(* PLC project LMM.project, Inovance company InoProShop(V1.9.1.6) InoProShop(V1.9.1.6) *)
(* stored: creationDateTime 2026-07-22T21:08:52.4325602, modificationDateTime 2026-07-22T21:08:38.7942337 *)

VAR_GLOBAL  (* GVL *)
  StartBtn AT %IX1.6 : BOOL;  (* 【面板启动】AT %IX1.6 → HMI_xStart/HMI_xEnable（上升沿 STOP→RUN） *)
  StopBtn AT %IX1.4 : BOOL;  (* 【面板停止】AT %IX1.4 → HMI_xStop *)
  ResetBtn : BOOL;  (* 【面板复位】→ HMI_xStopHold3s（错误复位脉冲）；地址现场可另绑 *)
  EStop AT %IX0.4 : BOOL;  (* 【面板急停】AT %IX0.4 正常=TRUE 按下=FALSE → 直通 HMI_xEStop *)
  StopLamp AT %QX0.6 : BOOL;  (* 【停止指示灯】AT %QX0.6 ← Dev_xStop（停止/待机） *)
  StartLamp AT %QX0.7 : BOOL;  (* 【启动/运行指示灯】AT %QX0.7 ← Dev_xRun（正在运行） *)
  JogVel : REAL;  (* 面板点动速度 → 桥接到 HMI_rJogVel* *)
  JogFwd : BOOL;  (* 面板前进 → 按 X 模式映射到 Sync/Diff/独立点动+ *)
  JogBwd : BOOL;  (* 面板后退 → 按 X 模式映射到 Sync/Diff/独立点动- *)
  JogUp : BOOL;  (* 面板上 → HMI_xJogZPos *)
  JogDown : BOOL;  (* 面板下 → HMI_xJogZNeg *)
  JogRight : BOOL;  (* 面板右 → HMI_xJogYPos *)
  JogLeft : BOOL;  (* 面板左 → HMI_xJogYNeg *)
  JogClockAdd : BOOL;  (* 顺时针 *)
  JogClockMis : BOOL;  (* 逆时针 *)
  JogACC : REAL;  (* 点动加速度 → AxisCmd_rAcc *)
  JogDEC : REAL;  (* 点动减速度 → AxisCmd_rDec *)
  HomeReq : BOOL;  (* 面板回零 → HMI_xHomeReqY/Z *)
  CaliForReq : BOOL;  (* 重力标定 *)
  ClearBruch : BOOL;  (* 毛刷清洗 *)
  yLength : REAL;  (* 龙门跨距/Y长度设定 4..6m → HMI_rWheelBase *)
  HMI_xEStop : BOOL;  (* 【急停】TRUE=未按下(正常)；FALSE=急停按下。可按可松，锁存由Logic保持 *)
  HMI_xStop : BOOL;  (* 【设备停止】短按RUN→STOP；长按3s故障复位 *)
  HMI_xStopHold3s : BOOL;  (* 【停止长按满3s脉冲】清急停锁存+轴错误复位+下使能 *)
  HMI_xEnable : BOOL;  (* 【使能/启动别名】与HMI_xStart等效；上升沿STOP→RUN *)
  Dev_xError : BOOL;  (* 【内部故障态】 *)
  Dev_xRun : BOOL;  (* 【内部运行态】 *)
  Dev_xStop : BOOL;  (* 【内部停机态】 *)
  eDevState : INT;  (* 【废弃】不做控制；显示请用 HMI_eDevState 派生 *)
  HMI_xDevError : BOOL;  (* 【故障灯设备级】 *)
  HMI_xDevRun : BOOL;  (* 【运行灯】 *)
  HMI_xDevStop : BOOL;  (* 【停机灯】 *)
  HMI_eOpMode : INT;  (* 【运行方式】0手动 1自动；配合Run灯 *)
  HMI_eDevState : INT;  (* 【设备状态码】0=STOP 1=RUN 2=ERROR *)
  HMI_xStart : BOOL;  (* 【设备启动】瞬时；上升沿STOP→RUN *)
  HMI_xJogYPos : BOOL;  (* 【Y点动+】TRUE移动 FALSE暂停；受限位/Z忙 *)
  HMI_xJogYNeg : BOOL;  (* 【Y点动-】TRUE移动 FALSE暂停 *)
  HMI_xJogZPos : BOOL;  (* 【Z点动+】TRUE移动 FALSE暂停 *)
  HMI_xJogZNeg : BOOL;  (* 【Z点动-】TRUE移动 FALSE暂停 *)
  HMI_xJogRPos : BOOL;  (* 【R点动+】预留；M5未就绪无效 *)
  HMI_xJogRNeg : BOOL;  (* 【R点动-】预留 *)
  HMI_xHomeY : BOOL;  (* 【Y回零】电平/上升沿触发；或配合轴选择\r\n *)
  HMI_xHomeZ : BOOL;  (* 【Z回零】电平/上升沿触发；或配合轴选择\r\n *)
  HMI_xHomeR : BOOL;  (* 【R回零】电平/上升沿触发；或配合轴选择\r\n *)
  HMI_iHomeAxis : INT := 0;  (* 【回零轴选择】0无 1=Y 2=Z 3=R\r\n *)
  HMI_xHomeExec : BOOL;  (* 【回零执行】上升沿：对 HMI_iHomeAxis 选定轴启动回零\r\n *)
  HMI_rJogVelX : REAL := 0.4;  (* 【X点动速度】龙门X基速设定 *)
  AxisCmd_rSpinVel : REAL := 0.0;
  HMI_rJogVelR : REAL := 0.2;  (* 【R轴手动速度】 *)
  HMI_rSpinVel : REAL := 0.3;  (* 【X轴旋转速度】 *)
  HMI_rJogVelY : REAL := 0.4;  (* 【Y点动速度】 *)
  HMI_rJogVelZ : REAL := 0.4;  (* 【Z点动速度】 *)
  HMI_rWheelBase : REAL := 5.0;  (* 【龙门跨距=Y行程】单位m，合法范围4..6；自动Y走距用此值 *)
  xEStopLatched : BOOL;  (* 【急停锁存】按下急停置位；仅长按停止复位可清 *)
  xEnablePermit : BOOL;  (* 【废弃】已删除设备态许可互锁 *)
  xFaultAggregate : BOOL;  (* 【故障汇总】任轴Fault *)
  xIlk_BlockYPlus : BOOL;  (* 【联锁禁Y+】由Y+限位派生 *)
  xIlk_BlockYNeg : BOOL;  (* 【联锁禁Y-】由Y-限位派生 *)
  xIlk_BlockZPlus : BOOL;  (* 【联锁禁Z+】由Z+限位派生 *)
  xIlk_BlockZNeg : BOOL;  (* 【联锁禁Z-】由Z-限位派生 *)
  xIlk_BlockYWhenZ : BOOL;  (* 【Z动禁Y】Z运动中禁止Y点动 *)
  xM5Ready : BOOL := TRUE;  (* 【第5轴就绪】TRUE=启用 R(Axis_4)；FALSE=忽略R\r\n *)
  HMI_xLampEStop : BOOL;  (* 【急停灯】HMI读；锁存或按钮仍按下 *)
  HMI_xLampEnableOk : BOOL;  (* 【使能/运行灯】=设备RUN *)
  HMI_xLampFault : BOOL;  (* 【轴故障灯】 *)
  eOpMode : INT;  (* 【运行模式】0=手动Manual（本期固定） *)
  iAlarmID : INT;  (* 【内部报警号】Logic判定后拷贝到HMI_iAlarmShow *)
  HMI_iAlarmShow : INT;  (* 【报警号】0无；1001急停；1002故障；1003限位；1004无许可；1099R未就绪 *)
  I_xLimYPos : BOOL;  (* 【Y正限位】物理输入，地址%I* TBD *)
  I_xLimYNeg : BOOL;  (* 【Y负限位】物理输入 *)
  I_xHomeY : BOOL;  (* 【Y原点】物理输入 *)
  I_xLimZPos : BOOL;  (* 【Z正限位】物理输入 *)
  I_xLimZNeg : BOOL;  (* 【Z负限位】物理输入 *)
  I_xHomeZ : BOOL;  (* 【Z原点】物理输入 *)
  I_xLimRPos : BOOL;  (* 【R正限位】预留 *)
  I_xLimRNeg : BOOL;  (* 【R负限位】预留 *)
  I_xHomeR : BOOL;  (* 【R原点】预留 *)
  AxisCmd_xPower : BOOL;  (* 【轴使能命令】仅设备RUN时TRUE *)
  AxisCmd_xJogYPos : BOOL;  (* 【Y点动+命令】含限位/Z忙门控 *)
  AxisCmd_xJogYNeg : BOOL;  (* 【Y点动-命令】 *)
  AxisCmd_xJogZPos : BOOL;  (* 【Z点动+命令】 *)
  AxisCmd_xJogZNeg : BOOL;  (* 【Z点动-命令】 *)
  AxisCmd_xJogRPos : BOOL;  (* 【R点动+命令】预留 *)
  AxisCmd_xJogRNeg : BOOL;  (* 【R点动-命令】预留 *)
  AxisCmd_xHomeY : BOOL;  (* 【Y回零】Logic→Axis；完成/停止后清\r\n *)
  AxisCmd_xHomeZ : BOOL;  (* 【Z回零】Logic→Axis；完成/停止后清\r\n *)
  AxisCmd_xHomeR : BOOL;  (* 【R回零】Logic→Axis；完成/停止后清\r\n *)
  AxisCmd_xStopAll : BOOL;  (* 【全停】急停/停止/故障时TRUE *)
  AxisCmd_xResetFault : BOOL;  (* 【错误复位脉冲】一拍TRUE→各轴MC_Reset *)
  AxisCmd_rWheelBase : REAL;  (* 【跨距L命令】限幅4..6m *)
  AxisCmd_rJogVelX : REAL;  (* 【X点动速度命令】 *)
  AxisCmd_rJogVelY : REAL;  (* 【Y点动速度命令】 *)
  AxisCmd_rJogVelZ : REAL;  (* 【Z点动速度命令】 *)
  AxisCmd_rJogVelR : REAL;  (* 【R点动速度命令】预留 *)
  AxisCmd_rAcc : REAL;  (* 【加速度】 *)
  AxisCmd_rDec : REAL;  (* 【减速度】 *)
  AxisFb_rVelCmdM1 : REAL;  (* 【M1速度指令反馈】供HMI显示 *)
  AxisFb_rVelCmdM2 : REAL;  (* 【M2速度指令反馈】 *)
  AxisFb_rPosM1 : REAL;  (* 【M1实际位置】 *)
  AxisFb_rPosM2 : REAL;  (* 【M2实际位置】 *)
  AxisFb_rPosY : REAL;  (* 【Y实际位置】 *)
  AxisFb_rPosZ : REAL;  (* 【Z实际位置】 *)
  AxisFb_rPosR : REAL;  (* 【R实际位置】预留 *)
  AxisFb_xStandstill1 : BOOL;  (* 【M1静止】 *)
  AxisFb_xStandstill2 : BOOL;  (* 【M2静止】 *)
  AxisFb_xStandstillY : BOOL;  (* 【Y静止】 *)
  AxisFb_xStandstillZ : BOOL;  (* 【Z静止】 *)
  AxisFb_xStandstillR : BOOL;  (* 【R静止】预留 *)
  AxisFb_xMovingM1 : BOOL;  (* 【M1运动中】 *)
  AxisFb_xMovingM2 : BOOL;  (* 【M2运动中】 *)
  AxisFb_xMovingY : BOOL;  (* 【Y运动中】 *)
  AxisFb_xMovingZ : BOOL;  (* 【Z运动中】 *)
  AxisFb_xMovingR : BOOL;  (* 【R运动中】预留 *)
  AxisFb_xPoweredM1 : BOOL;  (* 【M1已使能】驱动功率级就绪，HMI灯 *)
  AxisFb_xPoweredM2 : BOOL;  (* 【M2已使能】 *)
  AxisFb_xPoweredY : BOOL;  (* 【Y已使能】 *)
  AxisFb_xPoweredZ : BOOL;  (* 【Z已使能】 *)
  AxisFb_xPoweredR : BOOL;  (* 【R已使能】预留 *)
  AxisFb_xHomedY : BOOL;  (* 【Y已回零】 *)
  AxisFb_xHomedZ : BOOL;  (* 【Z已回零】 *)
  AxisFb_xHomedR : BOOL;  (* 【R已回零】Axis_4/_MC_Axis[5] *)
  AxisFb_xFaultM1 : BOOL;  (* 【M1故障】 *)
  AxisFb_xFaultM2 : BOOL;  (* 【M2故障】 *)
  AxisFb_xFaultY : BOOL;  (* 【Y故障】 *)
  AxisFb_xFaultZ : BOOL;  (* 【Z故障】 *)
  AxisFb_xFaultR : BOOL;  (* 【R故障】预留 *)
  AxisFb_xReady : BOOL;  (* 【轴就绪】四轴无故障、可参与运动 *)
  HMI_xAutoMode : BOOL;  (* 【自动模式】TRUE自动 FALSE手动 *)
  HMI_xJogXPos : BOOL;  (* 【X+】同步直行 *)
  HMI_xJogXNeg : BOOL;  (* 【X-】 *)
  HMI_xSpinLeft : BOOL;  (* 【左旋转】 *)
  HMI_xSpinRight : BOOL;  (* 【右旋转】 *)
  HMI_xAutoStart : BOOL;  (* 【自动启动】 *)
  HMI_xAutoAbort : BOOL;  (* 【自动中止】 *)
  HMI_rAutoDistX : REAL;  (* 【自动X距离】 *)
  HMI_rAutoVelX : REAL;  (* 【自动X速度】 *)
  HMI_rAutoVelY : REAL;  (* 【自动Y速度】 *)
  HMI_rAutoVelZ : REAL;  (* 【自动Z速度】 *)
  HMI_rForceSet : REAL;  (* 目标力设定(N)，力引导/自动压下用 *)
  HMI_xForceSimEnable : BOOL;  (* 力模拟使能：TRUE用HMI_rForceSim *)
  HMI_rForceSim : REAL;  (* 模拟力设定(N)，仅模拟使能时有效 *)
  HMI_iAutoStepShow : INT;  (* 【自动步号】 *)
  HMI_xAutoBusy : BOOL;  (* 【自动忙】 *)
  HMI_xAutoDone : BOOL;  (* 【自动完成】 *)
  HMI_rForceShow : REAL;  (* 力显示值(N)，供HMI/Web *)
  HMI_xHomedY : BOOL;  (* 【Y已回零】← AxisFb_xHomedY\r\n *)
  HMI_xHomedZ : BOOL;  (* 【Z已回零】← AxisFb_xHomedZ\r\n *)
  HMI_xHomedR : BOOL;  (* 【R已回零】← AxisFb_xHomedR\r\n *)
  HMI_xHomeBusyY : BOOL;  (* 【Y回零中】\r\n *)
  HMI_xHomeBusyZ : BOOL;  (* 【Z回零中】\r\n *)
  HMI_xHomeBusyR : BOOL;  (* 【R回零中】\r\n *)
  MB_CmdIn AT %IW103 : ARRAY[0..63] OF WORD;  (* Modbus TCP FC03 命令快照 Holding 1000..1063 *)
  MB_StatusOut AT %QW44 : ARRAY[0..63] OF WORD;  (* Modbus TCP FC16 状态快照 Holding 1100..1163 *)
  Tcp_iCommStatus : INT;  (* 0离线 1在线 2版本错误 3序号错误 4超时 *)
  Tcp_wLastHb : WORD;
  Tcp_wLastSeq : WORD;
  Tcp_wStatusSeq : WORD;
  Tcp_rKpTrack : REAL;
  Tcp_rKpForce : REAL;
  Tcp_xConnected : BOOL;  (* 【TCP】已连接 *)
  Tcp_xTimeout : BOOL;  (* 【TCP】通讯超时 *)
  Tcp_xOnline : BOOL;  (* 【TCP】Connected且未超时 *)
  Tcp_xEStop : BOOL := TRUE;  (* 【TCP急停影子】默认TRUE；与面板AND合成 *)
  Tcp_xStop : BOOL;
  Tcp_xStopHold3s : BOOL;
  Tcp_xStart : BOOL;
  Tcp_xEnable : BOOL;
  Tcp_xAutoMode : BOOL;
  Tcp_xJogXPos : BOOL;
  Tcp_xJogXNeg : BOOL;
  Tcp_xSpinLeft : BOOL;
  Tcp_xSpinRight : BOOL;
  Tcp_xJogYPos : BOOL;
  Tcp_xJogYNeg : BOOL;
  Tcp_xJogZPos : BOOL;
  Tcp_xJogZNeg : BOOL;
  Tcp_xJogRPos : BOOL;
  Tcp_xJogRNeg : BOOL;
  Tcp_xHomeY : BOOL;  (* TCP【Y回零】\r\n *)
  Tcp_xHomeZ : BOOL;  (* TCP【Z回零】\r\n *)
  Tcp_xHomeR : BOOL;  (* TCP【R回零】\r\n *)
  Tcp_iHomeAxis : INT := 0;  (* TCP【回零轴选择】0无 1=Y 2=Z 3=R\r\n *)
  Tcp_xHomeExec : BOOL;  (* TCP【回零执行】\r\n *)
  Tcp_rJogVelX : REAL := 0.4;
  Tcp_rSpinVel : REAL := 0.3;
  Tcp_rJogVelY : REAL := 0.3;
  Tcp_rJogVelZ : REAL := 0.2;
  Tcp_rJogVelR : REAL := 0.2;
  Tcp_xAutoStart : BOOL;
  Tcp_xAutoAbort : BOOL;
  Tcp_rAutoDistX : REAL := 1.0;
  Tcp_rAutoVelX : REAL := 0.4;
  Tcp_rAutoVelY : REAL := 0.3;
  Tcp_rAutoVelZ : REAL := 0.15;
  Tcp_rWheelBase : REAL := 5.0;
  Tcp_rForceSet : REAL := 100.0;  (* TCP影子：目标力(N) *)
  Tcp_xForceSimEnable : BOOL := TRUE;  (* TCP影子：力模拟使能 *)
  Tcp_rForceSim : REAL;  (* TCP影子：模拟力(N) *)
  Tcp_xForceTare : BOOL;  (* TCP影子：去皮 *)
  Tcp_xForceUntare : BOOL;  (* TCP影子：取消去皮 *)
  Tcp_xForceGuide : BOOL;  (* TCP影子：力引导使能 *)
  Tcp_uiPort : UINT := 9100;  (* 【TCP监听端口】默认9100 *)
  iAutoStep : INT;  (* 【自动步】0Idle..5Done *)
  rForceAct : REAL;  (* 实际力(N)，力传感换算或模拟值 *)
  rForceKp : REAL;  (* 恒力比例增益Kp，力引导Z轴用 *)
  Force_xEnable : BOOL := TRUE;  (* 力传感通讯总使能；FALSE时关闭SM1001 *)
  Force_wInRaw AT %IW102 : WORD;  (* Modbus读通道映射：保持寄存器0x0000原始力值 *)
  Force_xReadTrig : BOOL;  (* 探测读触发；可绑通道上升沿，循环读可不绑 *)
  Force_wOutTare AT %QW42 : WORD;  (* Modbus写通道：寄存器0x0011去皮(1)/取消(2) *)
  Force_wOutUnit AT %QW43 : WORD := 5;  (* Modbus写通道：寄存器0x0002单位，5=牛顿N *)
  Force_rScale : REAL := 0.01;  (* 原始值倍率，默认0.01(百分位) *)
  HMI_xForceTare : BOOL;  (* 去皮触发(上升沿)，面板/外部 *)
  HMI_xForceUntare : BOOL;  (* 取消去皮触发(上升沿) *)
  HMI_xForceGuide : BOOL;  (* 力引导使能：TRUE持续跟力，FALSE停止 *)
  Force_xCommOk : BOOL;  (* 通讯成功(已收到读回文) *)
  Force_xTimeout : BOOL;  (* 通讯超时/失败标志 *)
  Force_xSlaveFail : BOOL;  (* SM1001使能探测失败3次，报警1006 *)
  Force_xTareBusy : BOOL;  (* 去皮命令发送中 *)
  Force_xTareDone : BOOL;  (* 去皮完成脉冲 *)
  Logic_xForceTare : BOOL;  (* 自动步内部去皮脉冲(PRG_Logic写) *)
  Force_iRaw : INT;  (* 有符号原始力计数 *)
  Force_iState : INT;  (* 力任务状态：0闲置1使能2发读3等回文4成功-2失败 *)
  AxisCmd_xJogXPos : BOOL;  (* 【Axis X+】 *)
  AxisCmd_xJogXNeg : BOOL;  (* 【Axis X-】 *)
  AxisCmd_xSpinLeft : BOOL;  (* 【Axis 左旋】 *)
  AxisCmd_xSpinRight : BOOL;  (* 【Axis 右旋】 *)
  AxisCmd_xMoveRelX : BOOL;  (* 【Axis X相对】 *)
  AxisCmd_rMoveDistX : REAL;  (* 【X相对距离】 *)
  AxisCmd_rMoveVelX : REAL;  (* 【X相对速度】 *)
  AxisCmd_xMoveRelY : BOOL;  (* 【Axis Y相对】 *)
  AxisCmd_rMoveDistY : REAL;  (* 【Y相对距离】 *)
  AxisCmd_rMoveVelY : REAL;  (* 【Y相对速度】 *)
  AxisCmd_rZVelCmd : REAL;  (* 【Z速度指令】 *)
  AxisCmd_xUseZVelCmd : BOOL;  (* 【使用Z速度指令】 *)
  AxisCmd_xHoldR : BOOL;  (* 【R保持】 *)
  AxisCmd_rRHoldPos : REAL;  (* 【R保持角】 *)
  AxisFb_xMoveDoneX : BOOL;  (* 【X相对到位】 *)
  AxisFb_xMoveDoneY : BOOL;  (* 【Y相对到位】 *)
  HMI_iAutoPasses : INT := 1;
  Tcp_iAutoPasses : INT := 1;
  HMI_rHeadingErr : REAL := 0.0;
  Tcp_rHeadingErr : REAL := 0.0;
  HMI_rKpTrack : REAL := 0.0;
  HMI_rKpForce : REAL := 1.0;
  HMI_xStartReq : BOOL;
  HMI_xStopReq : BOOL;
  HMI_xResetReq : BOOL;
  HMI_xEStopReq : BOOL := TRUE;
  HMI_xAutoStartReq : BOOL;
  HMI_xAutoAbortReq : BOOL;
  AxisCmd_rHeadingErr : REAL;
  AxisCmd_rTrackKp : REAL;
  AxisCmd_rForceSet : REAL;
  AxisCmd_rForceKp : REAL;
  AxisCmd_rForceVelMax : REAL;
  AxisCmd_rMoveAbsPosY : REAL;
  AxisCmd_xForceFollow : BOOL;
  AxisCmd_xMoveAbsY : BOOL;
  AxisFb_xReadyM1 : BOOL;
  AxisFb_xReadyM2 : BOOL;
  AxisFb_xReadyY : BOOL;
  AxisFb_xReadyZ : BOOL;
  AxisFb_xReadyR : BOOL;
END_VAR

PROGRAM PRG_Axis_Control
  VAR
    fbM1 : FB_Servo;
    fbM2 : FB_Servo;
    fbY : FB_Servo;
    fbZ : FB_Servo;
    fbR : FB_Servo;
    fbForce : FB_Force;
    fbFF : FB_ForceFollow;
    fbTrack : FB_XLineTrack;
    iTrackMode : INT;
    rXBase : REAL;
    rXStart : LREAL;
    xMoveRelXPrev : BOOL;
    xXVelActive : BOOL;
  END_VAR

            (* PRG_Axis_Control — 运动独立任务(ETHERCAT)。只读 AxisCmd_*，写 AxisFb_*/rForceAct *)

(* ===== 力传感转换（本 POU 拥有 rForceAct） ===== *)
fbForce(wRaw := Force_wInRaw, rScale := Force_rScale, xEnable := Force_xEnable,
	xTare := HMI_xForceTare OR Logic_xForceTare, xUntare := HMI_xForceUntare);
Force_iRaw := fbForce.iRaw;
Force_xCommOk := fbForce.xCommOk;
Force_xTimeout := fbForce.xTimeout;
IF NOT HMI_xForceSimEnable THEN
	rForceAct := fbForce.rForceN;
END_IF;

(* ===== X 直线纠偏 / 原地转 ===== *)
iTrackMode := 0;
rXBase := 0.0;
IF AxisCmd_xMoveRelX THEN
	iTrackMode := 1;
	rXBase := ABS(AxisCmd_rMoveVelX);
ELSIF AxisCmd_xSpinLeft THEN
	iTrackMode := 2;
ELSIF AxisCmd_xSpinRight THEN
	iTrackMode := 3;
ELSIF AxisCmd_xJogXPos THEN
	iTrackMode := 1;
	rXBase := ABS(AxisCmd_rJogVelX);
ELSIF AxisCmd_xJogXNeg THEN
	iTrackMode := 1;
	rXBase := -ABS(AxisCmd_rJogVelX);
END_IF;

IF AxisCmd_xMoveRelX AND NOT xMoveRelXPrev THEN
	rXStart := fbM1.rActPos;
	AxisFb_xMoveDoneX := FALSE;
END_IF;
xMoveRelXPrev := AxisCmd_xMoveRelX;
IF AxisCmd_xMoveRelX THEN
	IF ABS(fbM1.rActPos - rXStart) >= ABS(AxisCmd_rMoveDistX) THEN
		AxisFb_xMoveDoneX := TRUE;
	END_IF;
ELSE
	AxisFb_xMoveDoneX := FALSE;
END_IF;

xXVelActive := (iTrackMode <> 0) AND NOT (AxisCmd_xMoveRelX AND AxisFb_xMoveDoneX);

fbTrack(xEnable := AxisCmd_xPower, xStop := AxisCmd_xStopAll, eMode := iTrackMode,
	rBaseVel := rXBase, rSpinVel := AxisCmd_rSpinVel,
	rHeadingErr := AxisCmd_rHeadingErr, rKpTrack := AxisCmd_rTrackKp, rTrimMax := 0.2);

fbM1(Axis := Axis, xEnable := AxisCmd_xPower, xStop := AxisCmd_xStopAll, xResetFault := AxisCmd_xResetFault,
	xUseVelCmd := xXVelActive, rVelCmd := fbTrack.rVelM1, rAcc := AxisCmd_rAcc, rDec := AxisCmd_rDec);
fbM2(Axis := Axis_1, xEnable := AxisCmd_xPower, xStop := AxisCmd_xStopAll, xResetFault := AxisCmd_xResetFault,
	xUseVelCmd := xXVelActive, rVelCmd := fbTrack.rVelM2, rAcc := AxisCmd_rAcc, rDec := AxisCmd_rDec);

(* ===== Y：回零 > 绝对(归位) > 相对(横移) > 点动 ===== *)
fbY(Axis := Axis_2, xEnable := AxisCmd_xPower, xStop := AxisCmd_xStopAll, xResetFault := AxisCmd_xResetFault,
	xHome := AxisCmd_xHomeY,
	xMoveAbs := AxisCmd_xMoveAbsY, rTargetPos := AxisCmd_rMoveAbsPosY,
	xMoveRel := AxisCmd_xMoveRelY, rDist := AxisCmd_rMoveDistY,
	xJogPos := AxisCmd_xJogYPos, xJogNeg := AxisCmd_xJogYNeg, rJogVel := AxisCmd_rJogVelY,
	rVel := AxisCmd_rMoveVelY, rAcc := AxisCmd_rAcc, rDec := AxisCmd_rDec);
AxisFb_xMoveDoneY := fbY.xMoveRelDone;

(* ===== Z：力跟随速度 > 回零 > 点动 ===== *)
fbFF(rForceSet := AxisCmd_rForceSet, rForceAct := rForceAct, rKp := AxisCmd_rForceKp,
	rVelMax := AxisCmd_rForceVelMax, rDeadband := 0.5, rPosZ := fbZ.rActPos,
	xHomedZ := fbZ.xHomed, xEnable := AxisCmd_xForceFollow, xInvert := FALSE);
fbZ(Axis := Axis_3, xEnable := AxisCmd_xPower, xStop := AxisCmd_xStopAll, xResetFault := AxisCmd_xResetFault,
	xHome := AxisCmd_xHomeZ,
	xUseVelCmd := AxisCmd_xForceFollow, rVelCmd := fbFF.rZVelCmd,
	xJogPos := AxisCmd_xJogZPos, xJogNeg := AxisCmd_xJogZNeg, rJogVel := AxisCmd_rJogVelZ,
	rAcc := AxisCmd_rAcc, rDec := AxisCmd_rDec);

(* ===== R：回零 > 保持角(绝对) > 点动；M5 门控 ===== *)
fbR(Axis := Axis_4, xEnable := AxisCmd_xPower AND xM5Ready, xStop := AxisCmd_xStopAll, xResetFault := AxisCmd_xResetFault,
	xHome := AxisCmd_xHomeR,
	xMoveAbs := AxisCmd_xHoldR, rTargetPos := AxisCmd_rRHoldPos,
	xJogPos := AxisCmd_xJogRPos, xJogNeg := AxisCmd_xJogRNeg, rJogVel := AxisCmd_rJogVelR,
	rVel := AxisCmd_rJogVelR, rAcc := AxisCmd_rAcc, rDec := AxisCmd_rDec);

(* ===== 反馈回写 ===== *)
AxisFb_rVelCmdM1 := fbTrack.rVelM1;
AxisFb_rVelCmdM2 := fbTrack.rVelM2;
AxisFb_rPosM1 := fbM1.rActPos; AxisFb_rPosM2 := fbM2.rActPos;
AxisFb_rPosY := fbY.rActPos; AxisFb_rPosZ := fbZ.rActPos; AxisFb_rPosR := fbR.rActPos;
AxisFb_xMovingM1 := fbM1.xMoving; AxisFb_xMovingM2 := fbM2.xMoving;
AxisFb_xMovingY := fbY.xMoving; AxisFb_xMovingZ := fbZ.xMoving; AxisFb_xMovingR := fbR.xMoving;
AxisFb_xStandstill1 := fbM1.xStandstill; AxisFb_xStandstill2 := fbM2.xStandstill;
AxisFb_xStandstillY := fbY.xStandstill; AxisFb_xStandstillZ := fbZ.xStandstill; AxisFb_xStandstillR := fbR.xStandstill;
AxisFb_xPoweredM1 := fbM1.xPowered; AxisFb_xPoweredM2 := fbM2.xPowered;
AxisFb_xPoweredY := fbY.xPowered; AxisFb_xPoweredZ := fbZ.xPowered; AxisFb_xPoweredR := fbR.xPowered;
AxisFb_xReadyM1 := fbM1.xReady; AxisFb_xReadyM2 := fbM2.xReady;
AxisFb_xReadyY := fbY.xReady; AxisFb_xReadyZ := fbZ.xReady; AxisFb_xReadyR := fbR.xReady;
AxisFb_xHomedY := fbY.xHomed; AxisFb_xHomedZ := fbZ.xHomed; AxisFb_xHomedR := fbR.xHomed;
AxisFb_xFaultM1 := fbM1.xFault; AxisFb_xFaultM2 := fbM2.xFault;
AxisFb_xFaultY := fbY.xFault; AxisFb_xFaultZ := fbZ.xFault; AxisFb_xFaultR := fbR.xFault;
AxisFb_xReady := fbM1.xReady AND fbM2.xReady AND fbY.xReady AND fbZ.xReady AND (NOT xM5Ready OR fbR.xReady);

          
END_PROGRAM

PROGRAM PRG_Force485
  VAR
    iSlaveStep : INT;
    iSlaveTry : INT;
    tonSlave : TON;
    wSnap : WORD;
    wRawLast : WORD;
    xTarePrev : BOOL;
    xUntarePrev : BOOL;
    xUnitInit : BOOL;
    diRaw : DINT;
    rTmp : REAL;
    xTareReq : BOOL;
  END_VAR

            (*==============================================================================
 * PRG_Force485 — SM1001 使能 + 发读等回文（最多3次）+ 去皮/换算
 *
 * 流程（严格按需求）：
 *   1) 使能 Modbus 从站 SM1001
 *   2) 发送一次读（破坏 Force_wInRaw 快照，等组态 FC03 通道写回 = 有回文）
 *   3) 有回文 → Force_xCommOk，进入成功态，不再重试
 *   4) 无回文 → 关闭 SM1001，重新使能，再读
 *   5) 3 次均无回文 → Force_xSlaveFail / 报警 1006
 *
 * 组态：读通道 FC03 0x0000 → Force_wInRaw（循环或由 Force_xReadTrig 触发均可）
 *============================================================================*)

Force_xTareDone := FALSE;

IF NOT Force_xEnable THEN
	SM1001 := FALSE;
	Force_xReadTrig := FALSE;
	Force_xCommOk := FALSE;
	Force_xTimeout := FALSE;
	Force_xTareBusy := FALSE;
	Force_xSlaveFail := FALSE;
	Force_iState := 0;
	iSlaveStep := 0;
	iSlaveTry := 0;
	RETURN;
END_IF;

CASE iSlaveStep OF
	0: (* 准备：先关从站，再进入使能 *)
		IF iSlaveTry >= 3 THEN
			SM1001 := FALSE;
			Force_xReadTrig := FALSE;
			Force_xSlaveFail := TRUE;
			Force_xTimeout := TRUE;
			Force_xCommOk := FALSE;
			Force_iState := -2;
			iSlaveStep := 99;
		ELSE
			SM1001 := FALSE;
			Force_xReadTrig := FALSE;
			Force_xCommOk := FALSE;
			tonSlave(IN := FALSE);
			tonSlave(IN := TRUE, PT := T#200MS);
			Force_iState := 0;
			iSlaveStep := 1;
		END_IF;

	1: (* 关断保持 *)
		SM1001 := FALSE;
		Force_xReadTrig := FALSE;
		tonSlave();
		IF tonSlave.Q THEN
			tonSlave(IN := FALSE);
			iSlaveStep := 2;
		END_IF;

	2: (* ① 使能从站 *)
		SM1001 := TRUE;
		Force_xReadTrig := FALSE;
		iSlaveTry := iSlaveTry + 1;
		tonSlave(IN := FALSE);
		tonSlave(IN := TRUE, PT := T#100MS);
		Force_iState := 1;
		iSlaveStep := 3;

	3: (* 使能稳定后：② 发读命令（破坏快照 + 读触发） *)
		SM1001 := TRUE;
		tonSlave();
		IF tonSlave.Q THEN
			(* 破坏映射值：有回文时通道会写回真实寄存器 *)
			wSnap := Force_wInRaw XOR 16#FFFF;
			Force_wInRaw := wSnap;
			Force_xReadTrig := FALSE;
			tonSlave(IN := FALSE);
			tonSlave(IN := TRUE, PT := T#20MS);
			Force_iState := 2;
			iSlaveStep := 4;
		END_IF;

	4: (* 读触发上升沿 *)
		SM1001 := TRUE;
		tonSlave();
		IF tonSlave.Q THEN
			Force_xReadTrig := TRUE;
			tonSlave(IN := FALSE);
			tonSlave(IN := TRUE, PT := T#500MS);
			Force_iState := 3;
			iSlaveStep := 5;
		END_IF;

	5: (* ③ 等回文：Force_wInRaw 被总线写回且不等于破坏值 *)
		SM1001 := TRUE;
		Force_xReadTrig := TRUE;
		tonSlave();
		IF Force_wInRaw <> wSnap THEN
			(* 有回文 → 成功，不再尝试 *)
			Force_xReadTrig := FALSE;
			Force_xCommOk := TRUE;
			Force_xTimeout := FALSE;
			Force_xSlaveFail := FALSE;
			wRawLast := Force_wInRaw;
			Force_iState := 4;
			tonSlave(IN := FALSE);
			iSlaveStep := 10;
		ELSIF tonSlave.Q THEN
			(* 无回文 → 关从站，回到 0 重新使能 *)
			Force_xReadTrig := FALSE;
			SM1001 := FALSE;
			Force_xCommOk := FALSE;
			Force_iState := 5;
			tonSlave(IN := FALSE);
			iSlaveStep := 0;
		END_IF;

	10: (* 成功：保持使能，不再重试使能 *)
		SM1001 := TRUE;
		Force_xReadTrig := FALSE;
		Force_xCommOk := TRUE;
		Force_xTimeout := FALSE;
		IF Force_wInRaw <> wRawLast THEN
			wRawLast := Force_wInRaw;
		END_IF;

	99: (* 3 次失败；复位清 Force_xSlaveFail 后从 0 重来 *)
		SM1001 := FALSE;
		Force_xReadTrig := FALSE;
		IF Force_xSlaveFail THEN
			Force_xTimeout := TRUE;
			Force_xCommOk := FALSE;
		ELSE
			iSlaveTry := 0;
			Force_xTimeout := FALSE;
			iSlaveStep := 0;
		END_IF;
END_CASE;

(* ----- 原始值换算（成功后持续；探测中也换算便于监视） ----- *)
diRaw := DWORD_TO_DINT(WORD_TO_DWORD(Force_wInRaw));
IF diRaw > 32767 THEN
	diRaw := diRaw - 65536;
END_IF;
Force_iRaw := DINT_TO_INT(diRaw);
IF Force_rScale < 1.0E-12 THEN
	rTmp := INT_TO_REAL(Force_iRaw);
ELSE
	rTmp := INT_TO_REAL(Force_iRaw) * Force_rScale;
END_IF;
IF NOT HMI_xForceSimEnable AND iSlaveStep = 10 THEN
	rForceAct := rTmp;
END_IF;

IF NOT xUnitInit AND iSlaveStep = 10 THEN
	Force_wOutUnit := 5;
	xUnitInit := TRUE;
END_IF;

xTareReq := FALSE;
IF iSlaveStep = 10 THEN
	IF ((HMI_xForceTare OR Tcp_xForceTare OR Logic_xForceTare) AND NOT xTarePrev) THEN
		Force_wOutTare := 1;
		xTareReq := TRUE;
		Force_xTareDone := TRUE;
	END_IF;
	xTarePrev := HMI_xForceTare OR Tcp_xForceTare OR Logic_xForceTare;
	IF Tcp_xForceTare THEN
		Tcp_xForceTare := FALSE;
	END_IF;
	IF Logic_xForceTare THEN
		Logic_xForceTare := FALSE;
	END_IF;

	IF ((HMI_xForceUntare OR Tcp_xForceUntare) AND NOT xUntarePrev) THEN
		Force_wOutTare := 2;
		xTareReq := TRUE;
		Force_xTareDone := TRUE;
	END_IF;
	xUntarePrev := HMI_xForceUntare OR Tcp_xForceUntare;
	IF Tcp_xForceUntare THEN
		Tcp_xForceUntare := FALSE;
	END_IF;
END_IF;

Force_xTareBusy := xTareReq;

          
END_PROGRAM

PROGRAM PRG_TcpHmi
  VAR
    xInit : BOOL;
    eCtrlSrc : INT;
    xPanelOp : BOOL;
    xTcpOp : BOOL;
    xValid : BOOL;
    wMagic : WORD;
    wVersion : WORD;
    wSeqHead : WORD;
    wSeqTail : WORD;
    wHeartbeat : WORD;
    dwTmp : DWORD;
    diTmp : DINT;
    i : INT;
    tonHb : TON;
  END_VAR

            (* PRG_TcpHmi — Modbus TCP 过程映像编解码 + 控制源仲裁 *)
(* PLC=Master 读 Holding1000 / 写 Holding1100；Gateway=Server *)
IF NOT xInit THEN
	Tcp_xEStop := TRUE;
	Tcp_rJogVelX := 0.4; Tcp_rSpinVel := 0.3;
	Tcp_rJogVelY := 0.3; Tcp_rJogVelZ := 0.2; Tcp_rJogVelR := 0.2;
	Tcp_rAutoDistX := 1.0; Tcp_rAutoVelX := 0.4;
	Tcp_rAutoVelY := 0.3; Tcp_rAutoVelZ := 0.15;
	Tcp_rWheelBase := 5.0; Tcp_rForceSet := 100.0;
	Tcp_xForceSimEnable := FALSE;
	Tcp_iAutoPasses := 1;
	Tcp_rHeadingErr := 0.0;
	Tcp_rKpTrack := 0.0; Tcp_rKpForce := 1.0;
	Tcp_iCommStatus := 0;
	Tcp_wLastHb := 0; Tcp_wLastSeq := 16#FFFF; Tcp_wStatusSeq := 0;
	tonHb(IN := FALSE);
	xInit := TRUE;
END_IF;

(* ===== 命令快照解码 ===== *)
wMagic := MB_CmdIn[0];
wVersion := MB_CmdIn[1];
wSeqHead := MB_CmdIn[2];
wHeartbeat := MB_CmdIn[3];
wSeqTail := MB_CmdIn[63];
xValid := (wMagic = 19533) AND (wVersion = 256) AND (wSeqHead = wSeqTail);
IF xValid THEN
	Tcp_iCommStatus := 1;
	IF wHeartbeat <> Tcp_wLastHb THEN
		tonHb(IN := FALSE);
		tonHb(IN := TRUE, PT := T#1S);
		Tcp_wLastHb := wHeartbeat;
	END_IF;
	IF wSeqHead <> Tcp_wLastSeq THEN
		Tcp_wLastSeq := wSeqHead;
		Tcp_xEStop := (MB_CmdIn[4] AND 1) <> 0;
		Tcp_xStop := (MB_CmdIn[4] AND 2) <> 0;
		Tcp_xStopHold3s := (MB_CmdIn[4] AND 4) <> 0;
		Tcp_xStart := (MB_CmdIn[4] AND 8) <> 0;
		Tcp_xEnable := (MB_CmdIn[4] AND 16) <> 0;
		Tcp_xAutoMode := (MB_CmdIn[4] AND 32) <> 0;
		Tcp_xJogXPos := (MB_CmdIn[4] AND 64) <> 0;
		Tcp_xJogXNeg := (MB_CmdIn[4] AND 128) <> 0;
		Tcp_xSpinLeft := (MB_CmdIn[4] AND 256) <> 0;
		Tcp_xSpinRight := (MB_CmdIn[4] AND 512) <> 0;
		Tcp_xJogYPos := (MB_CmdIn[4] AND 1024) <> 0;
		Tcp_xJogYNeg := (MB_CmdIn[4] AND 2048) <> 0;
		Tcp_xJogZPos := (MB_CmdIn[4] AND 4096) <> 0;
		Tcp_xJogZNeg := (MB_CmdIn[4] AND 8192) <> 0;
		Tcp_xJogRPos := (MB_CmdIn[4] AND 16384) <> 0;
		Tcp_xJogRNeg := (MB_CmdIn[4] AND 32768) <> 0;
		Tcp_xHomeY := (MB_CmdIn[5] AND 1) <> 0;
		Tcp_xHomeZ := (MB_CmdIn[5] AND 2) <> 0;
		Tcp_xHomeR := (MB_CmdIn[5] AND 4) <> 0;
		Tcp_xHomeExec := (MB_CmdIn[5] AND 8) <> 0;
		Tcp_xAutoStart := (MB_CmdIn[5] AND 16) <> 0;
		Tcp_xAutoAbort := (MB_CmdIn[5] AND 32) <> 0;
		Tcp_xForceSimEnable := (MB_CmdIn[5] AND 64) <> 0;
		Tcp_xForceTare := (MB_CmdIn[5] AND 128) <> 0;
		Tcp_xForceUntare := (MB_CmdIn[5] AND 256) <> 0;
		Tcp_xForceGuide := (MB_CmdIn[5] AND 512) <> 0;
		Tcp_iHomeAxis := WORD_TO_INT(MB_CmdIn[6]);
		Tcp_iAutoPasses := WORD_TO_INT(MB_CmdIn[7]);
		dwTmp := SHL(WORD_TO_DWORD(MB_CmdIn[8]), 16) OR WORD_TO_DWORD(MB_CmdIn[9]);
		Tcp_rJogVelX := DINT_TO_REAL(DWORD_TO_DINT(dwTmp)) / 1000.0;
		dwTmp := SHL(WORD_TO_DWORD(MB_CmdIn[10]), 16) OR WORD_TO_DWORD(MB_CmdIn[11]);
		Tcp_rSpinVel := DINT_TO_REAL(DWORD_TO_DINT(dwTmp)) / 1000.0;
		dwTmp := SHL(WORD_TO_DWORD(MB_CmdIn[12]), 16) OR WORD_TO_DWORD(MB_CmdIn[13]);
		Tcp_rJogVelY := DINT_TO_REAL(DWORD_TO_DINT(dwTmp)) / 1000.0;
		dwTmp := SHL(WORD_TO_DWORD(MB_CmdIn[14]), 16) OR WORD_TO_DWORD(MB_CmdIn[15]);
		Tcp_rJogVelZ := DINT_TO_REAL(DWORD_TO_DINT(dwTmp)) / 1000.0;
		dwTmp := SHL(WORD_TO_DWORD(MB_CmdIn[16]), 16) OR WORD_TO_DWORD(MB_CmdIn[17]);
		Tcp_rJogVelR := DINT_TO_REAL(DWORD_TO_DINT(dwTmp)) / 1000.0;
		dwTmp := SHL(WORD_TO_DWORD(MB_CmdIn[18]), 16) OR WORD_TO_DWORD(MB_CmdIn[19]);
		Tcp_rAutoDistX := DINT_TO_REAL(DWORD_TO_DINT(dwTmp)) / 1000.0;
		dwTmp := SHL(WORD_TO_DWORD(MB_CmdIn[20]), 16) OR WORD_TO_DWORD(MB_CmdIn[21]);
		Tcp_rAutoVelX := DINT_TO_REAL(DWORD_TO_DINT(dwTmp)) / 1000.0;
		dwTmp := SHL(WORD_TO_DWORD(MB_CmdIn[22]), 16) OR WORD_TO_DWORD(MB_CmdIn[23]);
		Tcp_rAutoVelY := DINT_TO_REAL(DWORD_TO_DINT(dwTmp)) / 1000.0;
		dwTmp := SHL(WORD_TO_DWORD(MB_CmdIn[24]), 16) OR WORD_TO_DWORD(MB_CmdIn[25]);
		Tcp_rAutoVelZ := DINT_TO_REAL(DWORD_TO_DINT(dwTmp)) / 1000.0;
		dwTmp := SHL(WORD_TO_DWORD(MB_CmdIn[26]), 16) OR WORD_TO_DWORD(MB_CmdIn[27]);
		Tcp_rWheelBase := DINT_TO_REAL(DWORD_TO_DINT(dwTmp)) / 1000.0;
		dwTmp := SHL(WORD_TO_DWORD(MB_CmdIn[28]), 16) OR WORD_TO_DWORD(MB_CmdIn[29]);
		Tcp_rForceSet := DINT_TO_REAL(DWORD_TO_DINT(dwTmp)) / 100.0;
		dwTmp := SHL(WORD_TO_DWORD(MB_CmdIn[30]), 16) OR WORD_TO_DWORD(MB_CmdIn[31]);
		Tcp_rForceSim := DINT_TO_REAL(DWORD_TO_DINT(dwTmp)) / 100.0;
		dwTmp := SHL(WORD_TO_DWORD(MB_CmdIn[32]), 16) OR WORD_TO_DWORD(MB_CmdIn[33]);
		Tcp_rHeadingErr := DINT_TO_REAL(DWORD_TO_DINT(dwTmp)) / 1000.0;
		dwTmp := SHL(WORD_TO_DWORD(MB_CmdIn[34]), 16) OR WORD_TO_DWORD(MB_CmdIn[35]);
		Tcp_rKpTrack := DINT_TO_REAL(DWORD_TO_DINT(dwTmp)) / 1000.0;
		dwTmp := SHL(WORD_TO_DWORD(MB_CmdIn[36]), 16) OR WORD_TO_DWORD(MB_CmdIn[37]);
		Tcp_rKpForce := DINT_TO_REAL(DWORD_TO_DINT(dwTmp)) / 1000.0;
	END_IF;
ELSIF wMagic <> 0 AND wMagic <> 19533 THEN
	Tcp_iCommStatus := 2;
ELSIF wSeqHead <> wSeqTail THEN
	Tcp_iCommStatus := 3;
END_IF;
tonHb();
IF tonHb.Q OR Tcp_iCommStatus = 0 THEN
	Tcp_xTimeout := TRUE;
	Tcp_xConnected := FALSE;
	Tcp_xOnline := FALSE;
	IF tonHb.Q THEN Tcp_iCommStatus := 4; END_IF;
	Tcp_xJogXPos := FALSE; Tcp_xJogXNeg := FALSE;
	Tcp_xSpinLeft := FALSE; Tcp_xSpinRight := FALSE;
	Tcp_xJogYPos := FALSE; Tcp_xJogYNeg := FALSE;
	Tcp_xJogZPos := FALSE; Tcp_xJogZNeg := FALSE;
	Tcp_xJogRPos := FALSE; Tcp_xJogRNeg := FALSE;
	Tcp_xHomeY := FALSE; Tcp_xHomeZ := FALSE; Tcp_xHomeR := FALSE;
	Tcp_xHomeExec := FALSE;
	Tcp_xStart := FALSE; Tcp_xEnable := FALSE;
	Tcp_xAutoStart := FALSE;
	Tcp_xForceTare := FALSE; Tcp_xForceUntare := FALSE; Tcp_xForceGuide := FALSE;
	Tcp_xStop := TRUE;
	Tcp_xAutoAbort := TRUE;
	Tcp_xEStop := TRUE;
ELSE
	Tcp_xTimeout := FALSE;
	Tcp_xConnected := TRUE;
	Tcp_xOnline := TRUE;
END_IF;

(* ===== 状态快照编码 ===== *)
Tcp_wStatusSeq := Tcp_wStatusSeq + 1;
MB_StatusOut[0] := 19533;
MB_StatusOut[1] := 256;
MB_StatusOut[2] := Tcp_wStatusSeq;
MB_StatusOut[3] := Tcp_wLastSeq;
MB_StatusOut[4] := Tcp_wLastHb;
FOR i := 5 TO 62 DO MB_StatusOut[i] := 0; END_FOR;
MB_StatusOut[5] := INT_TO_WORD(Tcp_iCommStatus);
MB_StatusOut[6] := INT_TO_WORD(HMI_eDevState);
MB_StatusOut[7] := INT_TO_WORD(HMI_eOpMode);
MB_StatusOut[8] := INT_TO_WORD(HMI_iAlarmShow);
MB_StatusOut[9] := INT_TO_WORD(HMI_iAutoStepShow);
IF HMI_xDevStop THEN MB_StatusOut[10] := MB_StatusOut[10] OR 1; END_IF;
IF HMI_xDevRun THEN MB_StatusOut[10] := MB_StatusOut[10] OR 2; END_IF;
IF HMI_xDevError THEN MB_StatusOut[10] := MB_StatusOut[10] OR 4; END_IF;
IF HMI_xLampEStop THEN MB_StatusOut[10] := MB_StatusOut[10] OR 8; END_IF;
IF HMI_xLampEnableOk THEN MB_StatusOut[10] := MB_StatusOut[10] OR 16; END_IF;
IF HMI_xLampFault THEN MB_StatusOut[10] := MB_StatusOut[10] OR 32; END_IF;
IF HMI_xAutoBusy THEN MB_StatusOut[10] := MB_StatusOut[10] OR 64; END_IF;
IF HMI_xAutoDone THEN MB_StatusOut[10] := MB_StatusOut[10] OR 128; END_IF;
IF HMI_xHomedY THEN MB_StatusOut[10] := MB_StatusOut[10] OR 256; END_IF;
IF HMI_xHomedZ THEN MB_StatusOut[10] := MB_StatusOut[10] OR 512; END_IF;
IF HMI_xHomedR THEN MB_StatusOut[10] := MB_StatusOut[10] OR 1024; END_IF;
IF HMI_xHomeBusyY THEN MB_StatusOut[10] := MB_StatusOut[10] OR 2048; END_IF;
IF HMI_xHomeBusyZ THEN MB_StatusOut[10] := MB_StatusOut[10] OR 4096; END_IF;
IF HMI_xHomeBusyR THEN MB_StatusOut[10] := MB_StatusOut[10] OR 8192; END_IF;
IF Tcp_xConnected THEN MB_StatusOut[10] := MB_StatusOut[10] OR 16384; END_IF;
IF Tcp_xTimeout THEN MB_StatusOut[10] := MB_StatusOut[10] OR 32768; END_IF;
IF Force_xCommOk THEN MB_StatusOut[11] := MB_StatusOut[11] OR 1; END_IF;
IF Force_xTimeout THEN MB_StatusOut[11] := MB_StatusOut[11] OR 2; END_IF;
IF Force_xSlaveFail THEN MB_StatusOut[11] := MB_StatusOut[11] OR 4; END_IF;
IF Force_xTareBusy THEN MB_StatusOut[11] := MB_StatusOut[11] OR 8; END_IF;
IF Force_xTareDone THEN MB_StatusOut[11] := MB_StatusOut[11] OR 16; END_IF;
IF AxisFb_xReady THEN MB_StatusOut[11] := MB_StatusOut[11] OR 32; END_IF;
IF AxisFb_xMoveDoneX THEN MB_StatusOut[11] := MB_StatusOut[11] OR 64; END_IF;
IF AxisFb_xMoveDoneY THEN MB_StatusOut[11] := MB_StatusOut[11] OR 128; END_IF;
IF AxisFb_xFaultM1 THEN MB_StatusOut[11] := MB_StatusOut[11] OR 256; END_IF;
IF AxisFb_xFaultM2 THEN MB_StatusOut[11] := MB_StatusOut[11] OR 512; END_IF;
IF AxisFb_xFaultY THEN MB_StatusOut[11] := MB_StatusOut[11] OR 1024; END_IF;
IF AxisFb_xFaultZ THEN MB_StatusOut[11] := MB_StatusOut[11] OR 2048; END_IF;
IF AxisFb_xFaultR THEN MB_StatusOut[11] := MB_StatusOut[11] OR 4096; END_IF;
IF AxisFb_xHomedY THEN MB_StatusOut[11] := MB_StatusOut[11] OR 8192; END_IF;
IF AxisFb_xHomedZ THEN MB_StatusOut[11] := MB_StatusOut[11] OR 16384; END_IF;
IF AxisFb_xHomedR THEN MB_StatusOut[11] := MB_StatusOut[11] OR 32768; END_IF;
diTmp := REAL_TO_DINT(HMI_rForceShow * 100.0);
dwTmp := DINT_TO_DWORD(diTmp);
MB_StatusOut[12] := DWORD_TO_WORD(SHR(dwTmp, 16));
MB_StatusOut[13] := DWORD_TO_WORD(dwTmp AND 16#FFFF);
diTmp := REAL_TO_DINT(AxisFb_rPosM1 * 1000.0);
dwTmp := DINT_TO_DWORD(diTmp);
MB_StatusOut[14] := DWORD_TO_WORD(SHR(dwTmp, 16));
MB_StatusOut[15] := DWORD_TO_WORD(dwTmp AND 16#FFFF);
diTmp := REAL_TO_DINT(AxisFb_rPosM2 * 1000.0);
dwTmp := DINT_TO_DWORD(diTmp);
MB_StatusOut[16] := DWORD_TO_WORD(SHR(dwTmp, 16));
MB_StatusOut[17] := DWORD_TO_WORD(dwTmp AND 16#FFFF);
diTmp := REAL_TO_DINT(AxisFb_rPosY * 1000.0);
dwTmp := DINT_TO_DWORD(diTmp);
MB_StatusOut[18] := DWORD_TO_WORD(SHR(dwTmp, 16));
MB_StatusOut[19] := DWORD_TO_WORD(dwTmp AND 16#FFFF);
diTmp := REAL_TO_DINT(AxisFb_rPosZ * 1000.0);
dwTmp := DINT_TO_DWORD(diTmp);
MB_StatusOut[20] := DWORD_TO_WORD(SHR(dwTmp, 16));
MB_StatusOut[21] := DWORD_TO_WORD(dwTmp AND 16#FFFF);
diTmp := REAL_TO_DINT(AxisFb_rPosR * 1000.0);
dwTmp := DINT_TO_DWORD(diTmp);
MB_StatusOut[22] := DWORD_TO_WORD(SHR(dwTmp, 16));
MB_StatusOut[23] := DWORD_TO_WORD(dwTmp AND 16#FFFF);
diTmp := REAL_TO_DINT(AxisFb_rVelCmdM1 * 1000.0);
dwTmp := DINT_TO_DWORD(diTmp);
MB_StatusOut[24] := DWORD_TO_WORD(SHR(dwTmp, 16));
MB_StatusOut[25] := DWORD_TO_WORD(dwTmp AND 16#FFFF);
diTmp := REAL_TO_DINT(AxisFb_rVelCmdM2 * 1000.0);
dwTmp := DINT_TO_DWORD(diTmp);
MB_StatusOut[26] := DWORD_TO_WORD(SHR(dwTmp, 16));
MB_StatusOut[27] := DWORD_TO_WORD(dwTmp AND 16#FFFF);
MB_StatusOut[63] := Tcp_wStatusSeq;

(* ===== 控制源仲裁（保留原语义） ===== *)
xPanelOp := StartBtn OR StopBtn OR ResetBtn OR JogFwd OR JogBwd OR JogLeft OR JogRight
	OR JogUp OR JogDown OR JogClockAdd OR JogClockMis;
xTcpOp := Tcp_xOnline AND (
	Tcp_xStart OR Tcp_xStop OR Tcp_xStopHold3s OR Tcp_xAutoStart OR Tcp_xAutoAbort
	OR Tcp_xJogXPos OR Tcp_xJogXNeg OR Tcp_xSpinLeft OR Tcp_xSpinRight
	OR Tcp_xJogYPos OR Tcp_xJogYNeg OR Tcp_xJogZPos OR Tcp_xJogZNeg
	OR Tcp_xJogRPos OR Tcp_xJogRNeg
	OR Tcp_xHomeY OR Tcp_xHomeZ OR Tcp_xHomeR OR Tcp_xHomeExec
	OR Tcp_xForceGuide OR Tcp_xForceTare OR Tcp_xForceUntare);
IF NOT Tcp_xOnline THEN
	eCtrlSrc := 0;
ELSIF xTcpOp THEN
	eCtrlSrc := 1;
ELSIF xPanelOp THEN
	eCtrlSrc := 0;
END_IF;

IF eCtrlSrc = 1 THEN
	HMI_xAutoMode := Tcp_xAutoMode;
	HMI_xJogXPos := Tcp_xJogXPos;   HMI_xJogXNeg := Tcp_xJogXNeg;
	HMI_xSpinLeft := Tcp_xSpinLeft; HMI_xSpinRight := Tcp_xSpinRight;
	HMI_xJogYPos := Tcp_xJogYPos;   HMI_xJogYNeg := Tcp_xJogYNeg;
	HMI_xJogZPos := Tcp_xJogZPos;   HMI_xJogZNeg := Tcp_xJogZNeg;
	HMI_xJogRPos := Tcp_xJogRPos;   HMI_xJogRNeg := Tcp_xJogRNeg;
	HMI_xHomeY := Tcp_xHomeY; HMI_xHomeZ := Tcp_xHomeZ; HMI_xHomeR := Tcp_xHomeR;
	HMI_iHomeAxis := Tcp_iHomeAxis; HMI_xHomeExec := Tcp_xHomeExec;
	HMI_xForceGuide := Tcp_xForceGuide;
	HMI_xForceTare := Tcp_xForceTare; HMI_xForceUntare := Tcp_xForceUntare;
	HMI_xForceSimEnable := Tcp_xForceSimEnable;
	HMI_rJogVelX := Tcp_rJogVelX; HMI_rSpinVel := Tcp_rSpinVel;
	HMI_rJogVelY := Tcp_rJogVelY; HMI_rJogVelZ := Tcp_rJogVelZ; HMI_rJogVelR := Tcp_rJogVelR;
	HMI_rAutoDistX := Tcp_rAutoDistX; HMI_rAutoVelX := Tcp_rAutoVelX;
	HMI_rAutoVelY := Tcp_rAutoVelY; HMI_rAutoVelZ := Tcp_rAutoVelZ;
	HMI_rWheelBase := Tcp_rWheelBase; HMI_rForceSet := Tcp_rForceSet;
	HMI_rForceSim := Tcp_rForceSim;
	HMI_iAutoPasses := Tcp_iAutoPasses;
	HMI_rHeadingErr := Tcp_rHeadingErr;
	HMI_rKpTrack := Tcp_rKpTrack;
	HMI_rKpForce := Tcp_rKpForce;
END_IF;

HMI_xEStop := EStop AND Tcp_xEStop AND HMI_xEStopReq;
HMI_xStart := StartBtn OR HMI_xStartReq OR (Tcp_xOnline AND Tcp_xStart);
HMI_xEnable := HMI_xStart;
HMI_xStop := StopBtn OR HMI_xStopReq OR (Tcp_xOnline AND Tcp_xStop);
HMI_xStopHold3s := ResetBtn OR HMI_xResetReq OR (Tcp_xOnline AND Tcp_xStopHold3s);
HMI_xAutoStart := (Tcp_xOnline AND Tcp_xAutoStart) OR ((eCtrlSrc = 0) AND HMI_xAutoStartReq);
HMI_xAutoAbort := HMI_xAutoAbortReq OR (Tcp_xOnline AND Tcp_xAutoAbort);

          
END_PROGRAM

FUNCTION_BLOCK FB_XDiff
  VAR_INPUT
    eMode : INT;
    eDiffFunc : INT;
    xJogSyncPos : BOOL;
    xJogSyncNeg : BOOL;
    xJogDiffPos : BOOL;
    xJogDiffNeg : BOOL;
    xStop : BOOL;
    xEnable : BOOL;
    rJogVel : REAL;
    rDiffDelta : REAL;
    rTurnOmega : REAL;
    rWheelBase : REAL;
  END_VAR
  VAR_OUTPUT
    rVelCmdM1 : REAL;
    rVelCmdM2 : REAL;
    xActive : BOOL;
    xUsePairVel : BOOL;
    xWheelBaseOk : BOOL;
  END_VAR

            (*==============================================================================
 * FB_XDiff — 龙门 X 双驱速度合成（仅 Axis 任务内使用）
 * eMode: 0=独立  1=同步同速平移  2=差速（子功能见 eDiffFunc）
 * eDiffFunc: 0=纠偏  1=原地旋转(一正一反)  2=差速拐弯
 * 跨距 rWheelBase: 4..6 m；X 运动方向与 Y 垂直
 *============================================================================*)

(* 输出清零 *)
rVelCmdM1 := 0.0;
rVelCmdM2 := 0.0;
xUsePairVel := FALSE;
xActive := FALSE;
(* 跨距合法性 *)
xWheelBaseOk := (rWheelBase >= 4.0) AND (rWheelBase <= 6.0);

(* 未使能 / 停止 / 独立模式：不合成成对速度 *)
IF NOT xEnable OR xStop OR eMode = 0 THEN
	RETURN;
END_IF;

(* ---------- Sync：两侧同速，龙门沿 X 平移 ---------- *)
IF eMode = 1 THEN
	IF xJogSyncPos XOR xJogSyncNeg THEN
		xUsePairVel := TRUE;
		xActive := TRUE;
		IF xJogSyncPos THEN
			rVelCmdM1 := rJogVel;
		ELSE
			rVelCmdM1 := -rJogVel;
		END_IF;
		rVelCmdM2 := rVelCmdM1; (* 同速 *)
	END_IF;
	RETURN;
END_IF;

(* ---------- Diff：需有方向键 ---------- *)
IF NOT (xJogDiffPos XOR xJogDiffNeg) THEN
	RETURN;
END_IF;

(* 原地旋转 / 差速拐弯依赖合法跨距 *)
IF (eDiffFunc = 1 OR eDiffFunc = 2) AND NOT xWheelBaseOk THEN
	RETURN;
END_IF;

xUsePairVel := TRUE;
xActive := TRUE;

CASE eDiffFunc OF
	0: (* 纠偏：同向 V±Δ，扶正龙门 *)
		IF xJogDiffPos THEN
			rVelCmdM1 := rJogVel + rDiffDelta;
			rVelCmdM2 := rJogVel - rDiffDelta;
		ELSE
			rVelCmdM1 := -(rJogVel + rDiffDelta);
			rVelCmdM2 := -(rJogVel - rDiffDelta);
		END_IF;

	1: (* 原地旋转：M1/M2 一正一反，转角度 *)
		IF ABS(rTurnOmega) > 1.0E-6 THEN
			rVelCmdM1 := rTurnOmega * rWheelBase * 0.5;
		ELSE
			rVelCmdM1 := rJogVel;
		END_IF;
		rVelCmdM2 := -rVelCmdM1;
		IF xJogDiffNeg THEN
			rVelCmdM1 := -rVelCmdM1;
			rVelCmdM2 := -rVelCmdM2;
		END_IF;

	2: (* 差速拐弯：两侧同向为主，速度差，可边走边弯 *)
		IF ABS(rTurnOmega) > 1.0E-6 THEN
			rVelCmdM1 := rJogVel + rTurnOmega * rWheelBase * 0.5;
			rVelCmdM2 := rJogVel - rTurnOmega * rWheelBase * 0.5;
		ELSE
			rVelCmdM1 := rJogVel + rDiffDelta;
			rVelCmdM2 := rJogVel - rDiffDelta;
		END_IF;
		IF xJogDiffNeg THEN
			rVelCmdM1 := -rVelCmdM1;
			rVelCmdM2 := -rVelCmdM2;
		END_IF;

ELSE
	xUsePairVel := FALSE;
	xActive := FALSE;
END_CASE;

          
END_FUNCTION_BLOCK

PROGRAM PLC_PRG

            (* MainTask 入口：HMI 交互 -> 设备逻辑；Axis 在 ETHERCAT 任务独立运行 *)
PRG_TcpHmi();
PRG_Logic();

          
END_PROGRAM

PROGRAM PRG_Logic
  VAR
    tonHold : TON;
    tonReady : TON;
    xResetPulse : BOOL;
    xResetPrev : BOOL;
    xSafe : BOOL;
    xAutoStartPrev : BOOL;
    xAutoStartEdge : BOOL;
    rRHold : REAL;
    iPass : INT;
    xAutoTareSent : BOOL;
    xHomeTrigY : BOOL;
    xHomeTrigZ : BOOL;
    xHomeTrigR : BOOL;
    xHomeTrigYPrev : BOOL;
    xHomeTrigZPrev : BOOL;
    xHomeTrigRPrev : BOOL;
    xAnyHomeBusy : BOOL;
    xReadyAll : BOOL;
  END_VAR

            (* PRG_Logic — 消费已仲裁 HMI_*；写 AxisCmd_*；状态只读派生（无状态机耦合） *)

(* 急停锁存 / 长按复位 *)
IF NOT HMI_xEStop THEN
	xEStopLatched := TRUE;
END_IF;
tonHold(IN := HMI_xStop AND HMI_xEStop, PT := T#3S);
xResetPulse := (HMI_xStopHold3s OR tonHold.Q) AND NOT xResetPrev;
xResetPrev := HMI_xStopHold3s OR tonHold.Q;
IF xResetPulse THEN
	xEStopLatched := FALSE;
	AxisCmd_xResetFault := TRUE;
	iAutoStep := 0;
	iPass := 0;
	Force_xSlaveFail := FALSE;
ELSE
	AxisCmd_xResetFault := FALSE;
END_IF;

(* 故障汇总：仅各轴 Errorstop *)
xFaultAggregate := AxisFb_xFaultM1 OR AxisFb_xFaultM2 OR AxisFb_xFaultY OR AxisFb_xFaultZ
	OR (xM5Ready AND AxisFb_xFaultR);

IF HMI_xAutoMode THEN eOpMode := 1; ELSE eOpMode := 0; END_IF;
HMI_eOpMode := eOpMode;

(* 安全 / 使能 —— 去耦：只看急停 + 故障 *)
xSafe := HMI_xEStop AND NOT xEStopLatched;
AxisCmd_xPower := xSafe;
AxisCmd_xStopAll := HMI_xStop OR NOT xSafe OR xFaultAggregate OR HMI_xAutoAbort;

(* 力/纠偏参数下发 *)
rForceKp := HMI_rKpForce;
IF rForceKp < 1.0E-6 THEN rForceKp := 1.0; END_IF;
AxisCmd_rForceSet := HMI_rForceSet;
AxisCmd_rForceKp := rForceKp;
AxisCmd_rForceVelMax := ABS(HMI_rAutoVelZ);
IF AxisCmd_rForceVelMax < 1.0E-6 THEN AxisCmd_rForceVelMax := ABS(HMI_rJogVelZ); END_IF;
AxisCmd_rHeadingErr := HMI_rHeadingErr;

IF HMI_xForceSimEnable THEN
	rForceAct := HMI_rForceSim;
END_IF;
HMI_rForceShow := rForceAct;

AxisCmd_rJogVelX := HMI_rJogVelX;
AxisCmd_rSpinVel := HMI_rSpinVel;
AxisCmd_rJogVelY := HMI_rJogVelY;
AxisCmd_rJogVelZ := HMI_rJogVelZ;
AxisCmd_rJogVelR := HMI_rJogVelR;
AxisCmd_rWheelBase := LIMIT(4.0, HMI_rWheelBase, 6.0);
AxisCmd_rAcc := JogACC;
AxisCmd_rDec := JogDEC;
IF AxisCmd_rAcc < 1.0 THEN AxisCmd_rAcc := 100.0; END_IF;
IF AxisCmd_rDec < 1.0 THEN AxisCmd_rDec := 100.0; END_IF;

(* 限位联锁；Z 回零后软限位 [-0.7,0] *)
xIlk_BlockYPlus := I_xLimYPos;
xIlk_BlockYNeg := I_xLimYNeg;
xIlk_BlockZPlus := I_xLimZPos OR (AxisFb_xHomedZ AND (AxisFb_rPosZ >= 0.0));
xIlk_BlockZNeg := I_xLimZNeg OR (AxisFb_xHomedZ AND (AxisFb_rPosZ <= -0.7));

(* 每拍清命令 *)
AxisCmd_xJogXPos := FALSE; AxisCmd_xJogXNeg := FALSE;
AxisCmd_xSpinLeft := FALSE; AxisCmd_xSpinRight := FALSE;
AxisCmd_xJogYPos := FALSE; AxisCmd_xJogYNeg := FALSE;
AxisCmd_xJogZPos := FALSE; AxisCmd_xJogZNeg := FALSE;
AxisCmd_xJogRPos := FALSE; AxisCmd_xJogRNeg := FALSE;
AxisCmd_xForceFollow := FALSE;
AxisCmd_xMoveRelX := FALSE;
AxisCmd_xMoveRelY := FALSE;
AxisCmd_xMoveAbsY := FALSE;
AxisCmd_xHoldR := FALSE;
AxisCmd_rTrackKp := 0.0;
Logic_xForceTare := FALSE;

xAutoStartEdge := HMI_xAutoStart AND NOT xAutoStartPrev;
xAutoStartPrev := HMI_xAutoStart;

IF HMI_xAutoAbort OR NOT xSafe OR xFaultAggregate THEN
	iAutoStep := 0;
	iPass := 0;
	HMI_xAutoBusy := FALSE;
END_IF;

(* ===== 手动 ===== *)
IF xSafe AND (eOpMode = 0) AND NOT HMI_xStop AND NOT xFaultAggregate THEN
	IF HMI_xSpinLeft XOR HMI_xSpinRight THEN
		AxisCmd_xSpinLeft := HMI_xSpinLeft;
		AxisCmd_xSpinRight := HMI_xSpinRight;
	ELSIF HMI_xJogXPos XOR HMI_xJogXNeg THEN
		AxisCmd_xJogXPos := HMI_xJogXPos;
		AxisCmd_xJogXNeg := HMI_xJogXNeg;
	END_IF;
	AxisCmd_xJogYPos := HMI_xJogYPos AND NOT xIlk_BlockYPlus;
	AxisCmd_xJogYNeg := HMI_xJogYNeg AND NOT xIlk_BlockYNeg;
	IF HMI_xForceGuide THEN
		AxisCmd_xForceFollow := TRUE;
	ELSE
		AxisCmd_xJogZPos := HMI_xJogZPos AND NOT xIlk_BlockZPlus;
		AxisCmd_xJogZNeg := HMI_xJogZNeg AND NOT xIlk_BlockZNeg;
	END_IF;
	IF xM5Ready THEN
		AxisCmd_xJogRPos := HMI_xJogRPos;
		AxisCmd_xJogRNeg := HMI_xJogRNeg;
	END_IF;
END_IF;

(* ===== 自动多道循环 ===== *)
IF xSafe AND (eOpMode = 1) AND NOT HMI_xStop AND NOT xFaultAggregate THEN
	IF iAutoStep = 0 AND xAutoStartEdge THEN
		rRHold := AxisFb_rPosR;
		xAutoTareSent := FALSE;
		HMI_xAutoDone := FALSE;
		HMI_xAutoBusy := TRUE;
		iPass := 1;
		iAutoStep := 1;
	END_IF;

	CASE iAutoStep OF
		1:
			AxisCmd_xHoldR := TRUE;
			AxisCmd_rRHoldPos := rRHold;
			AxisCmd_rTrackKp := HMI_rKpTrack;
			AxisCmd_rMoveDistX := HMI_rAutoDistX;
			AxisCmd_rMoveVelX := HMI_rAutoVelX;
			AxisCmd_xMoveRelX := TRUE;
			IF AxisFb_xMoveDoneX THEN
				AxisCmd_xMoveRelX := FALSE;
				iAutoStep := 2;
			END_IF;
		2:
			AxisCmd_xHoldR := TRUE;
			AxisCmd_rRHoldPos := rRHold;
			AxisCmd_rMoveAbsPosY := 0.0;
			AxisCmd_rMoveVelY := HMI_rAutoVelY;
			AxisCmd_xMoveAbsY := TRUE;
			IF AxisFb_xStandstillY AND (ABS(AxisFb_rPosY) < 0.005) THEN
				AxisCmd_xMoveAbsY := FALSE;
				xAutoTareSent := FALSE;
				iAutoStep := 3;
			END_IF;
		3:
			AxisCmd_xHoldR := TRUE;
			AxisCmd_rRHoldPos := rRHold;
			IF NOT xAutoTareSent THEN
				Logic_xForceTare := TRUE;
				xAutoTareSent := TRUE;
			END_IF;
			AxisCmd_xForceFollow := TRUE;
			IF rForceAct >= HMI_rForceSet THEN
				iAutoStep := 4;
			END_IF;
		4:
			AxisCmd_xHoldR := TRUE;
			AxisCmd_rRHoldPos := rRHold;
			AxisCmd_xForceFollow := TRUE;
			AxisCmd_rMoveDistY := AxisCmd_rWheelBase;
			AxisCmd_rMoveVelY := HMI_rAutoVelY;
			AxisCmd_xMoveRelY := TRUE;
			IF AxisFb_xMoveDoneY THEN
				AxisCmd_xMoveRelY := FALSE;
				iAutoStep := 5;
			END_IF;
		5:
			IF iPass < HMI_iAutoPasses THEN
				iPass := iPass + 1;
				iAutoStep := 1;
			ELSE
				iAutoStep := 6;
			END_IF;
		6:
			HMI_xAutoBusy := FALSE;
			HMI_xAutoDone := TRUE;
			iAutoStep := 0;
			iPass := 0;
	END_CASE;
END_IF;

(* ===== 回零：Y/Z/R；同时只回一轴 ===== *)
xHomeTrigY := HMI_xHomeY OR ((HMI_iHomeAxis = 1) AND HMI_xHomeExec);
xHomeTrigZ := HMI_xHomeZ OR ((HMI_iHomeAxis = 2) AND HMI_xHomeExec);
xHomeTrigR := HMI_xHomeR OR ((HMI_iHomeAxis = 3) AND HMI_xHomeExec);
xAnyHomeBusy := AxisCmd_xHomeY OR AxisCmd_xHomeZ OR AxisCmd_xHomeR;

IF AxisCmd_xStopAll OR NOT xSafe OR xFaultAggregate THEN
	AxisCmd_xHomeY := FALSE;
	AxisCmd_xHomeZ := FALSE;
	AxisCmd_xHomeR := FALSE;
ELSE
	IF AxisCmd_xHomeY AND AxisFb_xHomedY THEN AxisCmd_xHomeY := FALSE; END_IF;
	IF AxisCmd_xHomeZ AND AxisFb_xHomedZ THEN AxisCmd_xHomeZ := FALSE; END_IF;
	IF AxisCmd_xHomeR AND AxisFb_xHomedR THEN AxisCmd_xHomeR := FALSE; END_IF;
	IF (eOpMode = 0) AND NOT HMI_xStop THEN
		IF xHomeTrigY AND NOT xHomeTrigYPrev AND NOT xAnyHomeBusy THEN
			AxisCmd_xHomeY := TRUE;
		ELSIF xHomeTrigZ AND NOT xHomeTrigZPrev AND NOT xAnyHomeBusy THEN
			AxisCmd_xHomeZ := TRUE;
		ELSIF xHomeTrigR AND NOT xHomeTrigRPrev AND NOT xAnyHomeBusy AND xM5Ready THEN
			AxisCmd_xHomeR := TRUE;
		END_IF;
	END_IF;
END_IF;
xHomeTrigYPrev := xHomeTrigY;
xHomeTrigZPrev := xHomeTrigZ;
xHomeTrigRPrev := xHomeTrigR;

IF AxisCmd_xHomeY THEN AxisCmd_xJogYPos := FALSE; AxisCmd_xJogYNeg := FALSE; END_IF;
IF AxisCmd_xHomeZ THEN AxisCmd_xJogZPos := FALSE; AxisCmd_xJogZNeg := FALSE; AxisCmd_xForceFollow := FALSE; END_IF;
IF AxisCmd_xHomeR THEN AxisCmd_xJogRPos := FALSE; AxisCmd_xJogRNeg := FALSE; END_IF;

HMI_xHomedY := AxisFb_xHomedY;
HMI_xHomedZ := AxisFb_xHomedZ;
HMI_xHomedR := AxisFb_xHomedR;
HMI_xHomeBusyY := AxisCmd_xHomeY;
HMI_xHomeBusyZ := AxisCmd_xHomeZ;
HMI_xHomeBusyR := AxisCmd_xHomeR;

(* 使能就绪诊断 → 1007 *)
xReadyAll := AxisFb_xReadyM1 AND AxisFb_xReadyM2 AND AxisFb_xReadyY AND AxisFb_xReadyZ
	AND (NOT xM5Ready OR AxisFb_xReadyR);
tonReady(IN := AxisCmd_xPower AND NOT xReadyAll AND NOT xFaultAggregate, PT := T#2S);

(* 报警 *)
IF xEStopLatched OR NOT HMI_xEStop THEN
	iAlarmID := 1001;
ELSIF xFaultAggregate THEN
	iAlarmID := 1002;
ELSIF tonReady.Q THEN
	iAlarmID := 1007;
ELSIF NOT HMI_xForceSimEnable AND Force_xSlaveFail THEN
	iAlarmID := 1006;
ELSIF NOT HMI_xForceSimEnable AND Force_xTimeout THEN
	iAlarmID := 1005;
ELSE
	iAlarmID := 0;
END_IF;

(* 状态灯（只读派生，不互锁） *)
Dev_xError := xFaultAggregate;
Dev_xRun := xSafe AND NOT HMI_xStop AND NOT xFaultAggregate;
Dev_xStop := NOT Dev_xRun AND NOT Dev_xError;
HMI_xDevError := Dev_xError;
HMI_xDevRun := Dev_xRun;
HMI_xDevStop := Dev_xStop;
IF Dev_xError THEN HMI_eDevState := 2;
ELSIF Dev_xRun THEN HMI_eDevState := 1;
ELSE HMI_eDevState := 0; END_IF;

HMI_iAutoStepShow := iAutoStep;
HMI_xLampEStop := xEStopLatched OR NOT HMI_xEStop;
HMI_xLampEnableOk := Dev_xRun;
HMI_xLampFault := xFaultAggregate;
HMI_iAlarmShow := iAlarmID;

StopLamp := Dev_xStop;
StartLamp := Dev_xRun;

          
END_PROGRAM

FUNCTION_BLOCK FB_Servo
  VAR_INPUT
    xEnable : BOOL;
    xJogPos : BOOL;
    xJogNeg : BOOL;
    xStop : BOOL;
    xResetFault : BOOL;
    xHome : BOOL;
    xUseVelCmd : BOOL;
    rVelCmd : REAL;
    rJogVel : REAL;
    xMoveRel : BOOL;
    rDist : REAL;
    xMoveAbs : BOOL;
    rTargetPos : REAL;
    rVel : REAL;
    rAcc : REAL;
    rDec : REAL;
  END_VAR
  VAR_OUTPUT
    xPowered : BOOL;
    xReady : BOOL;
    xMoving : BOOL;
    xStandstill : BOOL;
    xHomed : BOOL;
    xFault : BOOL;
    xMoveRelDone : BOOL;
    xMoveAbsDone : BOOL;
    rActPos : LREAL;
  END_VAR
  VAR_IN_OUT
    Axis : AXIS_REF_SM3;
  END_VAR
  VAR
    fbPower : MC_Power;
    fbJog : MC_MoveVelocity;
    fbStop : MC_Stop;
    fbHome : MC_Home;
    fbReset : MC_Reset;
    fbReadStatus : MC_ReadStatus;
    fbReadPos : MC_ReadActualPosition;
    fbSetPos : MC_SetPosition;
    fbMoveRel : MC_MoveRelative;
    fbMoveAbs : MC_MoveAbsolute;
    xEnInternal : BOOL;
    xHomePrev : BOOL;
    xZeroReq : BOOL;
  END_VAR

            (* FB_Servo — 单轴原子。仲裁：停止/故障 > 回零 > 绝对 > 相对 > 速度 > 点动 > 空闲 *)
fbReadStatus(Axis := Axis, Enable := TRUE);
fbReadPos(Axis := Axis, Enable := TRUE);
rActPos := fbReadPos.Position;
xStandstill := fbReadStatus.StandStill;
xMoving := fbReadStatus.DiscreteMotion OR fbReadStatus.ContinuousMotion;
xFault := fbReadStatus.Errorstop;

fbReset(Axis := Axis, Execute := xResetFault);

xEnInternal := xEnable AND NOT xStop AND NOT fbReadStatus.Errorstop;
fbPower(Axis := Axis, Enable := TRUE, bRegulatorOn := xEnInternal, bDriveStart := xEnInternal);
xPowered := fbPower.Status;
xReady := fbPower.Status AND NOT fbReadStatus.Errorstop;

IF xHome AND NOT xHomePrev THEN
	xHomed := FALSE;
	xZeroReq := FALSE;
END_IF;
xHomePrev := xHome;

IF xStop OR NOT xEnable OR fbReadStatus.Errorstop THEN
	fbMoveRel(Axis := Axis, Execute := FALSE);
	fbMoveAbs(Axis := Axis, Execute := FALSE);
	fbJog(Axis := Axis, Execute := FALSE);
	fbHome(Axis := Axis, Execute := FALSE, Position := 0.0);
	fbStop(Axis := Axis, Execute := TRUE, Deceleration := rDec);
	xZeroReq := FALSE;
	xMoveRelDone := FALSE;
	xMoveAbsDone := FALSE;

ELSIF xHome THEN
	fbStop(Axis := Axis, Execute := FALSE);
	fbJog(Axis := Axis, Execute := FALSE);
	fbMoveRel(Axis := Axis, Execute := FALSE);
	fbMoveAbs(Axis := Axis, Execute := FALSE);
	fbHome(Axis := Axis, Execute := TRUE, Position := 0.0);
	IF fbHome.Done THEN
		xZeroReq := TRUE;
	END_IF;

ELSIF xMoveAbs THEN
	fbStop(Axis := Axis, Execute := FALSE);
	fbJog(Axis := Axis, Execute := FALSE);
	fbHome(Axis := Axis, Execute := FALSE, Position := 0.0);
	fbMoveRel(Axis := Axis, Execute := FALSE);
	fbMoveAbs(Axis := Axis, Execute := xPowered, Position := rTargetPos,
		Velocity := ABS(rVel), Acceleration := rAcc, Deceleration := rDec);
	xMoveAbsDone := fbMoveAbs.Done;

ELSIF xMoveRel THEN
	fbStop(Axis := Axis, Execute := FALSE);
	fbJog(Axis := Axis, Execute := FALSE);
	fbHome(Axis := Axis, Execute := FALSE, Position := 0.0);
	fbMoveAbs(Axis := Axis, Execute := FALSE);
	fbMoveRel(Axis := Axis, Execute := xPowered, Distance := rDist,
		Velocity := ABS(rVel), Acceleration := rAcc, Deceleration := rDec);
	xMoveRelDone := fbMoveRel.Done;

ELSIF xUseVelCmd THEN
	fbStop(Axis := Axis, Execute := FALSE);
	fbHome(Axis := Axis, Execute := FALSE, Position := 0.0);
	fbMoveRel(Axis := Axis, Execute := FALSE);
	fbMoveAbs(Axis := Axis, Execute := FALSE);
	IF ABS(rVelCmd) > 1.0E-6 AND xPowered THEN
		fbJog(Axis := Axis, Execute := TRUE, Velocity := rVelCmd, Acceleration := rAcc, Deceleration := rDec);
	ELSE
		fbJog(Axis := Axis, Execute := FALSE);
	END_IF;

ELSIF xJogPos XOR xJogNeg THEN
	fbStop(Axis := Axis, Execute := FALSE);
	fbHome(Axis := Axis, Execute := FALSE, Position := 0.0);
	fbMoveRel(Axis := Axis, Execute := FALSE);
	fbMoveAbs(Axis := Axis, Execute := FALSE);
	IF xPowered THEN
		IF xJogPos THEN
			fbJog(Axis := Axis, Execute := TRUE, Velocity := ABS(rJogVel), Acceleration := rAcc, Deceleration := rDec);
		ELSE
			fbJog(Axis := Axis, Execute := TRUE, Velocity := -ABS(rJogVel), Acceleration := rAcc, Deceleration := rDec);
		END_IF;
	ELSE
		fbJog(Axis := Axis, Execute := FALSE);
	END_IF;

ELSE
	fbJog(Axis := Axis, Execute := FALSE);
	fbHome(Axis := Axis, Execute := FALSE, Position := 0.0);
	fbMoveRel(Axis := Axis, Execute := FALSE);
	fbMoveAbs(Axis := Axis, Execute := FALSE);
	fbStop(Axis := Axis, Execute := FALSE);
	xMoveRelDone := FALSE;
	xMoveAbsDone := FALSE;
END_IF;

fbSetPos(Axis := Axis, Execute := xZeroReq, Position := 0.0);
IF fbSetPos.Done THEN
	xHomed := TRUE;
	xZeroReq := FALSE;
END_IF;

          
END_FUNCTION_BLOCK

FUNCTION_BLOCK FB_Force
  VAR_INPUT
    wRaw : WORD;
    rScale : REAL;
    xEnable : BOOL;
    xTare : BOOL;
    xUntare : BOOL;
  END_VAR
  VAR_OUTPUT
    rForceN : REAL;
    iRaw : INT;
    xCommOk : BOOL;
    xTimeout : BOOL;
  END_VAR
  VAR
    rTare : REAL;
    xTarePrev : BOOL;
    xUntarePrev : BOOL;
    wPrev : WORD;
    tonStale : TON;
    rRawScaled : REAL;
  END_VAR

            (* FB_Force — Modbus 原始力换算 + 软件去皮 + 通讯看门狗（仅提示） *)
iRaw := WORD_TO_INT(wRaw);
rRawScaled := INT_TO_REAL(iRaw) * rScale;

IF xTare AND NOT xTarePrev THEN
	rTare := rRawScaled;
END_IF;
xTarePrev := xTare;
IF xUntare AND NOT xUntarePrev THEN
	rTare := 0.0;
END_IF;
xUntarePrev := xUntare;

rForceN := rRawScaled - rTare;

tonStale(IN := xEnable AND (wRaw = wPrev), PT := T#2S);
wPrev := wRaw;
xTimeout := xEnable AND tonStale.Q;
xCommOk := xEnable AND NOT xTimeout;

          
END_FUNCTION_BLOCK

FUNCTION_BLOCK FB_ForceFollow
  VAR_INPUT
    rForceSet : REAL;
    rForceAct : REAL;
    rKp : REAL;
    rVelMax : REAL;
    rDeadband : REAL;
    rPosZ : LREAL;
    xHomedZ : BOOL;
    xEnable : BOOL;
    xInvert : BOOL;
  END_VAR
  VAR_OUTPUT
    rZVelCmd : REAL;
    xInBand : BOOL;
  END_VAR
  VAR
    rErr : REAL;
    rV : REAL;
  END_VAR

            (* FB_ForceFollow — Z 恒力 P 控制律；向下=负；回零后夹紧 [-0.7,0] *)
IF NOT xEnable THEN
	rZVelCmd := 0.0;
	xInBand := FALSE;
	RETURN;
END_IF;

rErr := rForceSet - rForceAct;
rV := -rKp * rErr;
IF xInvert THEN
	rV := -rV;
END_IF;
rV := LIMIT(-ABS(rVelMax), rV, ABS(rVelMax));

xInBand := ABS(rErr) < rDeadband;
IF xInBand THEN
	rV := 0.0;
END_IF;

IF xHomedZ THEN
	IF (rPosZ >= 0.0) AND (rV > 0.0) THEN
		rV := 0.0;
	END_IF;
	IF (rPosZ <= -0.7) AND (rV < 0.0) THEN
		rV := 0.0;
	END_IF;
END_IF;

rZVelCmd := rV;

          
END_FUNCTION_BLOCK

FUNCTION_BLOCK FB_XLineTrack
  VAR_INPUT
    xEnable : BOOL;
    xStop : BOOL;
    eMode : INT;
    rBaseVel : REAL;
    rSpinVel : REAL;
    rHeadingErr : REAL;
    rKpTrack : REAL;
    rTrimMax : REAL;
  END_VAR
  VAR_OUTPUT
    rVelM1 : REAL;
    rVelM2 : REAL;
    xActive : BOOL;
  END_VAR
  VAR
    rTrim : REAL;
  END_VAR

            (* FB_XLineTrack — X 直行按航向角纠偏差速 / 原地左右转 *)
rTrim := LIMIT(-ABS(rTrimMax), rKpTrack * rHeadingErr, ABS(rTrimMax));

CASE eMode OF
	1:
		rVelM1 := rBaseVel + rTrim;
		rVelM2 := rBaseVel - rTrim;
	2:
		rVelM1 := ABS(rSpinVel);
		rVelM2 := -ABS(rSpinVel);
	3:
		rVelM1 := -ABS(rSpinVel);
		rVelM2 := ABS(rSpinVel);
ELSE
	rVelM1 := 0.0;
	rVelM2 := 0.0;
END_CASE;

IF xStop OR NOT xEnable THEN
	rVelM1 := 0.0;
	rVelM2 := 0.0;
END_IF;

xActive := (eMode <> 0) AND xEnable AND NOT xStop;

          
END_FUNCTION_BLOCK

CONFIGURATION Device
END_CONFIGURATION

CONFIGURATION HIGH_SPEED_IO
END_CONFIGURATION

CONFIGURATION ETHERCAT
END_CONFIGURATION

CONFIGURATION MDX_EC
END_CONFIGURATION

CONFIGURATION Axis
END_CONFIGURATION

CONFIGURATION MDX_EC_1
END_CONFIGURATION

CONFIGURATION Axis_1
END_CONFIGURATION

CONFIGURATION MDX_EC_2
END_CONFIGURATION

CONFIGURATION Axis_2
END_CONFIGURATION

CONFIGURATION MDX_EC_3
END_CONFIGURATION

CONFIGURATION Axis_3
END_CONFIGURATION

CONFIGURATION MDX_EC_4
END_CONFIGURATION

CONFIGURATION Axis_4
END_CONFIGURATION

CONFIGURATION MODBUS_COM0
END_CONFIGURATION

CONFIGURATION modbus_protocol
END_CONFIGURATION

CONFIGURATION MODBUS_TCP
END_CONFIGURATION

CONFIGURATION modbusTcp
END_CONFIGURATION
